// TIA Portal V19 export
TYPE "LAF_typeOperationInterlockProcessValues"
TITLE = LLGES_OperatorInterlockProcessValues
// Module related monitoring information
// stored: Access Published
   STRUCT
      maintenanceLockActive { ExternalWritable := 'False'} : Bool;   // TRUE: Maintenance lock is active, information to lock the HMI
   END_STRUCT;
END_TYPE
